{attribute 'qualified_only'}
VAR_GLOBAL
	temperature : REAL;
	Pressure : REAL;
	
	startCommand : BOOL;
	stopCommand : BOOL;
	
END_VAR

(* stored: Version 1.1.0.1, ProductVersion 3.1.4024.12
   GVL GVL_Test: Id {c1bbfc22-bd03-4efe-9a03-d02a5c4a7f1f} *)
